FUNCTION_BLOCK FB_MaintenanceCounter
VAR_INPUT
    bCountPulse      : BOOL;   
    bReset           : BOOL;   
    nLimit           : UDINT;  
END_VAR
VAR_OUTPUT
    nCurrentCount    : UDINT;  
    bMaintenanceDue  : BOOL;   
END_VAR
VAR
    fbRisingEdge     : R_TRIG; 
END_VAR


fbRisingEdge(CLK := bCountPulse);


IF fbRisingEdge.Q THEN
    nCurrentCount := nCurrentCount + 1;
END_IF

IF bReset THEN
    nCurrentCount := 0;
END_IF


bMaintenanceDue := (nCurrentCount >= nLimit) AND (nLimit > 0);

END_FUNCTION_BLOCK

(* stored: Version 1.1.0.1, ProductVersion 3.1.4024.16
   POU FB_MaintenanceCounter: Id {e845490c-d475-42d4-9822-5d76cb9b4e38}, SpecialFunc None *)
